{attribute 'linkalways'} 
{attribute 'no_explicit_call' := 'This FB is a CLASS and must be accessed using methods or properties'}
{attribute 'enable_dynamic_creation'}
FUNCTION_BLOCK SessionsMiddleware EXTENDS MiddlewareBase
VAR
	sessionManager: I_SessionManager;
	config : I_SessionMiddlewareConfig;
END_VAR

METHOD FB_init : BOOL
VAR_INPUT
	bInitRetains : BOOL; // if TRUE, the retain variables are initialized (warm start / cold start)
	bInCopyCode : BOOL;  // if TRUE, the instance afterwards gets moved into the copy code (online change)
	SessionManager : I_SessionManager;
	Config : I_SessionMiddlewareConfig;
END_VAR
THIS^.sessionManager := SessionManager;
THIS^.config := Config;
END_METHOD

METHOD PUBLIC Handle
VAR_INPUT
	Request : I_Request;
	Response : I_ServerResponse;
END_VAR
VAR
	sessionId : T_MAXSTRING;
END_VAR
IF (NOT config.TryGetSessionIdFromRequest(Request, sessionId)) OR_ELSE (NOT sessionManager.IsValidSession(sessionId)) THEN
	sessionId := sessionManager.CreateSession();
	config.UpdateRequestWithSessionId(Request,sessionId);
END_IF

sessionManager.RefreshSession(sessionId);

config.UpdateResponseWithSessionId(Response, sessionId);
Next(Request, Response);
END_METHOD

END_FUNCTION_BLOCK

(* stored: Version 1.1.0.1, ProductVersion 3.1.4024.12
   POU SessionsMiddleware: Id {d93490f3-dd35-4e22-a3f9-48c0397af766}, SpecialFunc None
   Folder Constructor: Id {05de603a-654d-42ee-aa4a-a59f76429878}
   Method FB_init: Id {70964f61-6718-48b9-b225-f89a36eb1cd6}
   Method Handle: Id {d2badea3-44aa-48aa-87d1-835b91359ac5} *)
